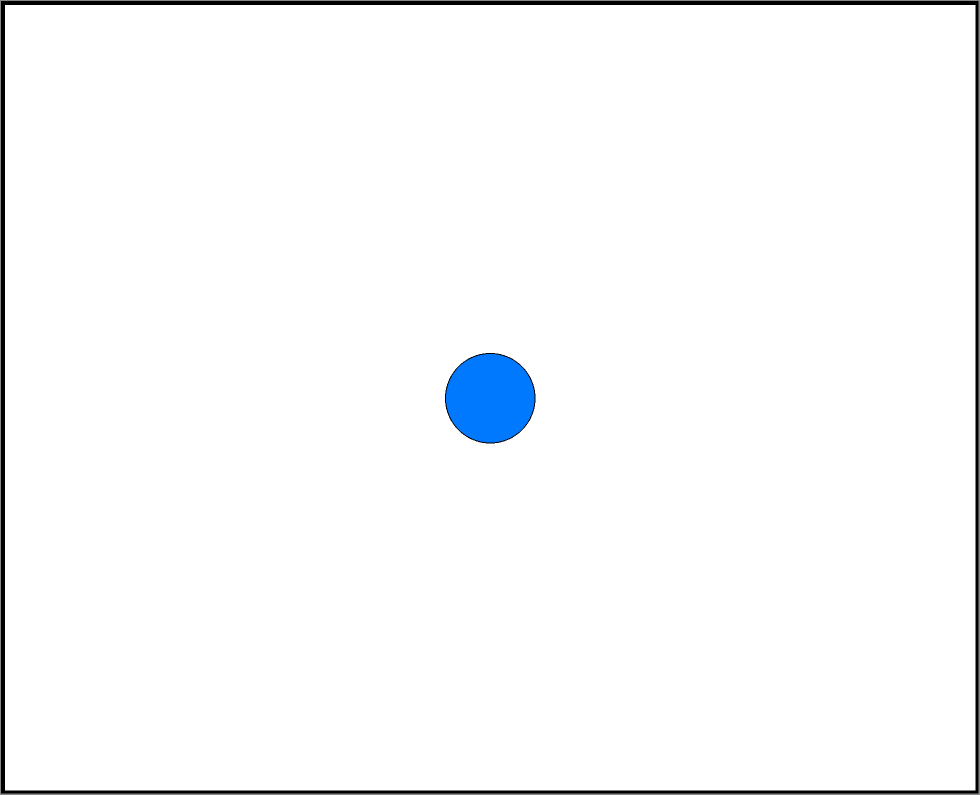
VISUALIZATION FigureGeneratorDisplay  // 980x795
    Rectangle (0,0 980x795)
    Frame (0,0 980x795)
        shows Polygon(pVisu := MAIN.FB_FigureGenerator.pVisu, VisuLenght := MAIN.FB_FigureGenerator.VisuLenght)
    Ellipse (445,353 90x90), invisible if: NOT Touchpanel.bContactAvailable
        p3560616238: Touchpanel.touch_scale_x.rX_mm*3
        p2738717112: -Touchpanel.touch_scale_y.rX_mm*3
END_VISUALIZATION

(* stored: Version 1.1.0.1, ProductVersion 3.1.4024.12
   Visu FigureGeneratorDisplay: Id {3145b3a2-a4fa-42f2-9fdc-3b573a7f6509} *)
